{attribute addProperty BoxType "EL1259-0000-0016"}
{attribute addProperty Id "Output_event_state_1BIT10.12533Output_event_state_2BIT10.12534Output_event_state_3BIT10.12535Output_event_state_4BIT10.12536Output_event_state_5BIT10.12537Output_event_state_6BIT10.12538Output_event_state_7BIT10.12539Output_event_state_8BIT10.12540Output_event_state_9BIT10.12541Output_event_state_10BIT10.12542"}
{attribute addProperty CRC "3258946073"}
{attribute addProperty SizeInBites "186"}
{attribute addProperty SizeInBytes "23.25"}
{warning 'Size of this structure is not a multiple of 8 bits!!!'}
TYPE Outputs_C23F9219 :
STRUCT
	{attribute addProperty Name "Output_event_state_1"}
	Output_event_state_1 : BIT;
	{attribute addProperty Name "Output_event_state_2"}
	Output_event_state_2 : BIT;
	{attribute addProperty Name "Output_event_state_3"}
	Output_event_state_3 : BIT;
	{attribute addProperty Name "Output_event_state_4"}
	Output_event_state_4 : BIT;
	{attribute addProperty Name "Output_event_state_5"}
	Output_event_state_5 : BIT;
	{attribute addProperty Name "Output_event_state_6"}
	Output_event_state_6 : BIT;
	{attribute addProperty Name "Output_event_state_7"}
	Output_event_state_7 : BIT;
	{attribute addProperty Name "Output_event_state_8"}
	Output_event_state_8 : BIT;
	{attribute addProperty Name "Output_event_state_9"}
	Output_event_state_9 : BIT;
	{attribute addProperty Name "Output_event_state_10"}
	Output_event_state_10 : BIT;
	{attribute 'hide'}
	reserve_3_BOOL_0 : BOOL;
	{attribute 'hide'}
	reserve_3_BOOL_1 : BOOL;
	{attribute 'hide'}
	reserve_3_BOOL_2 : BOOL;
	{attribute 'hide'}
	reserve_3_BOOL_3 : BOOL;
	{attribute 'hide'}
	reserve_3_BOOL_4 : BOOL;
	{attribute 'hide'}
	reserve_3_BOOL_5 : BOOL;
	{attribute 'hide'}
	reserve_3_BOOL_6 : BOOL;
	{attribute 'hide'}
	reserve_3_BOOL_7 : BOOL;
	{attribute 'hide'}
	reserve_3_BOOL_8 : BOOL;
	{attribute 'hide'}
	reserve_3_BOOL_9 : BOOL;
	{attribute 'hide'}
	reserve_3_BOOL_10 : BOOL;
	{attribute 'hide'}
	reserve_3_BOOL_11 : BOOL;
	{attribute 'hide'}
	reserve_3_BOOL_12 : BOOL;
	{attribute 'hide'}
	reserve_3_BOOL_13 : BOOL;
	{attribute 'hide'}
	reserve_3_BOOL_14 : BOOL;
	{attribute 'hide'}
	reserve_3_BOOL_15 : BOOL;
	{attribute 'hide'}
	reserve_3_BOOL_16 : BOOL;
	{attribute 'hide'}
	reserve_3_BOOL_17 : BOOL;
	{attribute 'hide'}
	reserve_3_BOOL_18 : BOOL;
	{attribute 'hide'}
	reserve_3_BOOL_19 : BOOL;
	{attribute 'hide'}
	reserve_3_BOOL_20 : BOOL;
	{attribute 'hide'}
	reserve_3_BOOL_21 : BOOL;
END_STRUCT
END_TYPE

(* stored: Version 1.2.0.0, ProductVersion 3.1.4024.9
   DUT Outputs_C23F9219: Id {92d982ec-f3a7-4fae-8cf7-de5ff29425b6} *)
